FUNCTION_BLOCK SludgeBufferStatus_2 (* Basic Function Block Type *)
  (* Standard: 61499-2 *)
  (* Version 0.0, 6/10/2026, Schneider Electric, Template *)
  PACKAGE SE.Nereda;
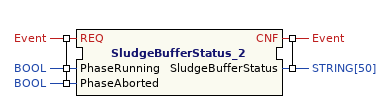
  EVENT_INPUT
    REQ WITH PhaseRunning, PhaseAborted; (* Normal Execution Request *)
  END_EVENT
  EVENT_OUTPUT
    CNF WITH SludgeBufferStatus; (* Execution Confirmation *)
  END_EVENT
  VAR_INPUT
    PhaseRunning : BOOL;
    PhaseAborted : BOOL;
  END_VAR
  VAR_OUTPUT
    SludgeBufferStatus : STRING[50]; (* Output event qualifier *)
  END_VAR
  VAR
    Init : BOOL;
  END_VAR
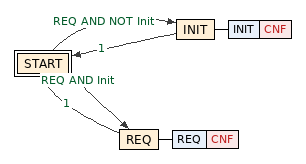
  EC_STATES
    START; (* Initial State *)
    REQ : REQ -> CNF; (* Normal execution *)
    INIT : INIT -> CNF;
  END_STATES
  EC_TRANSITIONS
    START TO REQ := REQ AND Init;
    REQ TO START := 1;
    START TO INIT := REQ AND NOT Init;
    INIT TO START := 1;
  END_TRANSITIONS
  ALGORITHM REQ IN ST: (* Normally executed algorithm *)
;
IF PhaseRunning AND NOT PhaseAborted THEN
	SludgeBufferStatus := 'SludgeBuffer Running';
ELSIF NOT PhaseRunning AND PhaseAborted THEN
	SludgeBufferStatus := 'SludgeBuffer Aborted';
ELSE
	SludgeBufferStatus := 'SludgeBuffer Status';
END_IF;
  END_ALGORITHM
  ALGORITHM INIT IN ST:
;
Init := TRUE;
SludgeBufferStatus := 'SludgeBuffer Status';
  END_ALGORITHM
END_FUNCTION_BLOCK
